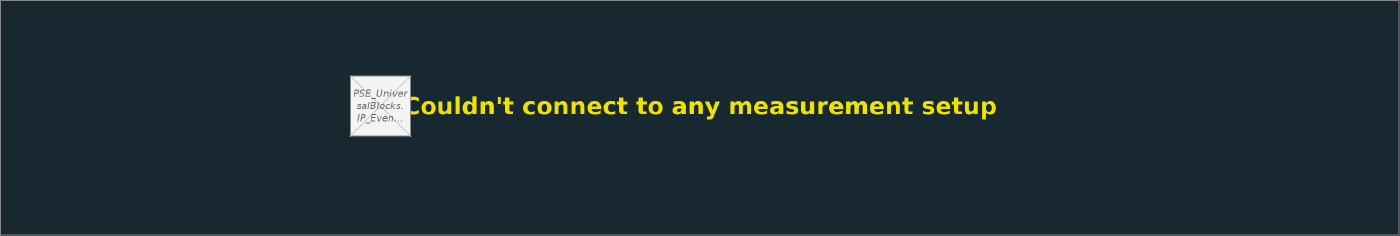
VISUALIZATION InitializingNoFixturesAvailable  // 1480x250
    Label (0,92 1480x40), "Couldn't connect to any measurement setup"
    Image (370,80 64x64), image: PSE_UniversalBlocks.IP_EventSeverity.critical
END_VISUALIZATION

(* stored: Version 1.1.0.1, ProductVersion 3.1.4024.9
   Visu InitializingNoFixturesAvailable: Id {743103fb-4885-4901-a7ef-67c618aee312} *)
